// TIA Portal V17 export
// export: Created 2022-02-03T14:45:10.6899411Z, ExportSetting WithDefaults, DisplayName Totally Integrated Automation Portal, DisplayVersion V17, DisplayName TIA Portal Openness, DisplayVersion V17, DisplayName TIA Portal Version Control Interface, DisplayVersion V17, DisplayName SINAMICS Startdrive Advanced, DisplayVersion V17, DisplayName SINAMICS Startdrive G130, G150, S120, S150, SINAMICS MV, S210, DisplayVersion V17, DisplayName SINAMICS Startdrive G110M, G120, G120C, G120D, G120P, G115D, DisplayVersion V17, DisplayName STEP 7 Professional, DisplayVersion V17, DisplayName STEP 7 Safety, DisplayVersion V17, DisplayName WinCC Advanced, DisplayVersion V17
FUNCTION_BLOCK "BayOccupied"   // FB3, LAD
VERSION : 0.1
// stored: Access Published, AutoNumber true, IsIECCheckEnabled false, IsRetainMemResEnabled false, MemoryReserve 100, SetENOAutomatically false, UDAEnableTagReadback false
   VAR_INPUT
      operationMode : Bool;
      conveyorLeft : Bool;
      bBay : Bool;
      sBay : Bool;
      currentStoreFull : Bool;
   END_VAR
   VAR_IN_OUT
      occupiedBay : Bool;
   END_VAR
   VAR
      staOldConveyorLeft : Bool;
   END_VAR
   VAR_TEMP   // added for the SCL form of the ladder/FBD networks
      _w1 : Bool;
      _w2 : Bool;
   END_VAR
BEGIN

REGION Network 1
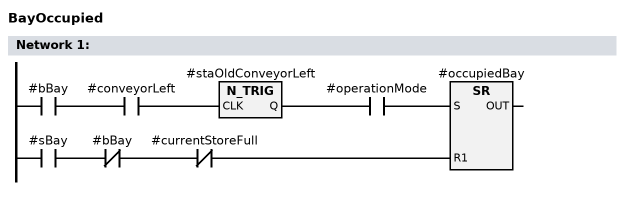
   RUNG wire#powerrail
      Contact( #bBay )
      Contact( #conveyorLeft )
      N_Trig( #staOldConveyorLeft )
      Contact( #operationMode )
      S_SR(operand := #occupiedBay, r1 := wire#w1)
   END_RUNG
   RUNG wire#powerrail
      Contact( #sBay )
      I_Contact( #bBay )
      I_Contact( #currentStoreFull )
   END_RUNG wire#w1
   // the same network as SCL:
   #_w1 := #bBay AND #conveyorLeft;
   #_w2 := NOT #_w1 AND #staOldConveyorLeft;   // falling edge
   #staOldConveyorLeft := #_w1;
   IF #_w2 AND #operationMode THEN
       #occupiedBay := TRUE;   // SR flip-flop
   END_IF;
   IF #sBay AND NOT #bBay AND NOT #currentStoreFull THEN #occupiedBay := FALSE; END_IF;
END_REGION
END_FUNCTION_BLOCK
